// Mitsubishi GX Works2 project: PLC_Group_44   PLC: FX3G

// global labels: Global1
VAR_GLOBAL
  switch7 AT X007 : BOOL;
  lamp7 AT Y007 : BOOL;
  berry_input AT D1100 : INT;
  lemon_input AT D1102 : INT;
  STABILIZER_input AT D1104 : INT;
  GUM_input AT D1106 : INT;
  BERRY_stock AT D1200 : INT;
  LEMON_stock AT D1202 : INT;
  STABILIZER_stock AT D1204 : INT;
  GUM_stock AT D1206 : INT;
  M_start AT M0 : BOOL;
  storage AT D1304 : INT;
  switch5 AT X005 : BOOL;
  analog_input1 AT D8280 : INT;
  switch1 AT X001 : BOOL;
  save_analog_input1 AT D8202 : INT;
END_VAR
VAR_GLOBAL CONSTANT
  K_5 : INT := 2000;
  K_6 : INT := 2400;
  K_10 : INT := 4000;
END_VAR
VAR_GLOBAL
  M_normal AT M1 : BOOL;
  M_pinuk AT M2 : BOOL;
END_VAR
VAR_GLOBAL CONSTANT
  K_7 : INT := 7;
  K_berry_normal : INT := 280;
  K_berry_pinuk : INT := 385;
  K_lemon_normal : INT := 455;
  K_lemon_pinuk : INT := 665;
  K_gum_normal : INT := 28;
  K_gum_pinuk : INT := 70;
  K_stabilizer_normal : INT := 105;
  K_stabilizer_pinuk : INT := 210;
END_VAR
VAR_GLOBAL
  M_exit AT M4 : BOOL;
  BERRY_to_subtract AT D1500 : INT;
  LEMON_to_subtract AT D1502 : INT;
  STABILIZER_to_subtract AT D1504 : INT;
  GUM_to_subtract AT D1506 : INT;
  M_check_stock AT M5 : BOOL;
  M_make_icecream AT M6 : BOOL;
END_VAR
VAR_GLOBAL CONSTANT
  K_berry_total_normal : INT := 350;
  K_berry_total_pinuk : INT := 560;
  K_lemon_total_normal : INT := 490;
  K_lemon_total_pinuk : INT := 700;
END_VAR
VAR_GLOBAL
  BERRY_total AT D1508 : INT;
  LEMON_total AT D1510 : INT;
  making_icecream_timer_c AT TC0 : BOOL;
END_VAR
VAR_GLOBAL CONSTANT
  K_50 : INT := 50;
END_VAR
VAR_GLOBAL
  making_icecream_timer_s AT TS0 : BOOL;
  lamp0 AT Y000 : BOOL;
  M_empty AT M7 : BOOL;
  M_cool_icecream AT M8 : BOOL;
  switch2 AT X002 : BOOL;
  cooling_icecream_timer_c AT TC1 : BOOL;
  cooling_icecream_timer_s AT TS1 : BOOL;
END_VAR
VAR_GLOBAL CONSTANT
  K_80 : INT := 80;
END_VAR
VAR_GLOBAL
  lamp2 AT Y002 : BOOL;
  switch3 AT X003 : BOOL;
  M_mix_materials AT M9 : BOOL;
  M_make_icecream_timer AT M11 : BOOL;
  M_cool_icecream_timer AT M10 : BOOL;
END_VAR
VAR_GLOBAL CONSTANT
  K_mixing_total_normal : INT := 868;
  K_mixing_total_pinuk : INT := 1330;
  K_3 : INT := 3;
END_VAR
VAR_GLOBAL
  mixing_total AT D1512 : INT;
  mixing_duration AT D1514 : INT;
  M_mix_materials_timer AT M12 : BOOL;
  mix_materials_timer_c AT TC2 : BOOL;
  mix_materials_timer_s AT TS2 : BOOL;
  lamp_5_timer_c AT TC3 : BOOL;
  lamp_5_timer_s AT TS3 : BOOL;
  lamp5 AT Y005 : BOOL;
  lamp_6_timer_c AT TC4 : BOOL;
  lamp_6_timer_s AT TS4 : BOOL;
  lamp6 AT Y006 : BOOL;
END_VAR
VAR_GLOBAL CONSTANT
  K_30 : INT := 30;
  K_01 : INT := 40;
  K_0 : INT;
END_VAR
VAR_GLOBAL
  M_BERRY_stock_check AT M14 : BOOL;
  M_LEMON_stock_check AT M15 : BOOL;
  M_STABILIZER_stock_check AT M16 : BOOL;
  M_GUM_stock_check AT M17 : BOOL;
  analog_output AT D8282 : INT;
END_VAR
VAR_GLOBAL CONSTANT
  K_10_timer : INT := 10;
END_VAR
VAR_GLOBAL
  M_cool_and_mix AT M18 : BOOL;
  make_LEMON AT D1308 : INT;
  make_BERRY AT D1306 : INT;
  cool_BERRY AT D1300 : INT;
  cool_LEMON AT D1302 : INT;
  mix_container AT D1310 : INT;
  M_blink_lamps AT M13 : BOOL;
  M_enough_stock AT M3 : BOOL;
END_VAR

// task Task_01 (event TRUE, interval 0, priority 31): POU_01

PROGRAM POU_01
(* structured ladder/FBD written out as ST: instructions are called as NAME(EN, inputs, outputs); _pN, _eN, _tN stand for wires *)
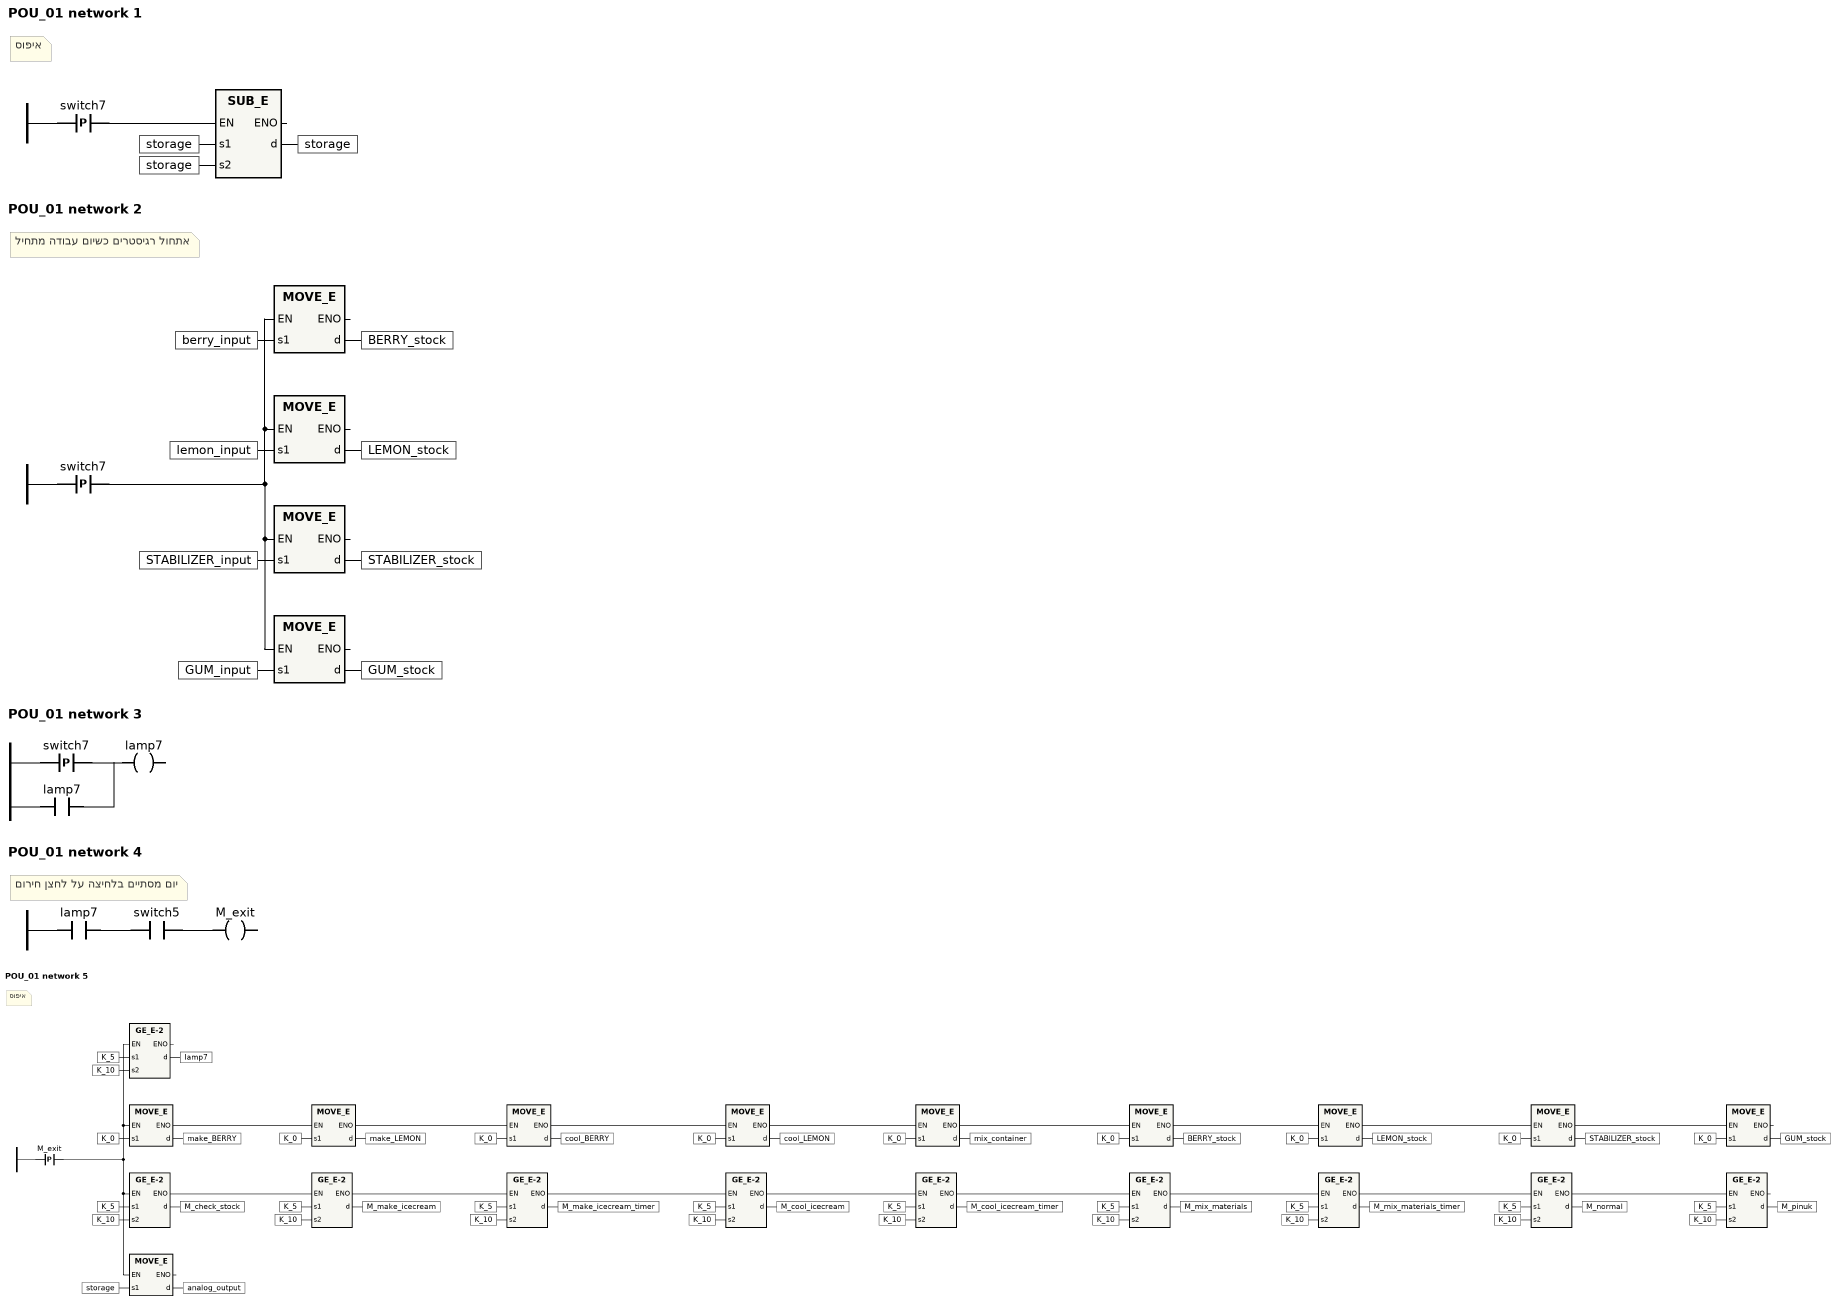
(* network 1 *)
(* איפוס *)
SUB_E(LDP(TRUE, switch7), storage, storage, storage);
(* network 2 *)
(* אתחול רגיסטרים כשיום עבודה מתחיל *)
_p1 := LDP(TRUE, switch7);
MOVE_E(_p1, berry_input, BERRY_stock);
MOVE_E(_p1, lemon_input, LEMON_stock);
MOVE_E(_p1, STABILIZER_input, STABILIZER_stock);
MOVE_E(_p1, GUM_input, GUM_stock);
(* network 3 *)
lamp7 := LDP(TRUE, switch7) OR lamp7;
(* network 4 *)
(* יום מסתיים בלחיצה על לחצן חירום *)
M_exit := lamp7 AND switch5;
(* network 5 *)
(* איפוס *)
_p1 := LDP(TRUE, M_exit);
GE_E(_p1, K_5, K_10, lamp7);
_e2 := MOVE_E(_p1, K_0, make_BERRY);
_e3 := MOVE_E(_e2, K_0, make_LEMON);
_e4 := MOVE_E(_e3, K_0, cool_BERRY);
_e5 := MOVE_E(_e4, K_0, cool_LEMON);
_e6 := MOVE_E(_e5, K_0, mix_container);
_e7 := MOVE_E(_e6, K_0, BERRY_stock);
_e8 := MOVE_E(_e7, K_0, LEMON_stock);
_e9 := MOVE_E(_e8, K_0, STABILIZER_stock);
MOVE_E(_e9, K_0, GUM_stock);
MOVE_E(_p1, storage, analog_output);
_e10 := GE_E(_p1, K_5, K_10, M_check_stock);
_e11 := GE_E(_e10, K_5, K_10, M_make_icecream);
_e12 := GE_E(_e11, K_5, K_10, M_make_icecream_timer);
_e13 := GE_E(_e12, K_5, K_10, M_cool_icecream);
_e14 := GE_E(_e13, K_5, K_10, M_cool_icecream_timer);
_e15 := GE_E(_e14, K_5, K_10, M_mix_materials);
_e16 := GE_E(_e15, K_5, K_10, M_mix_materials_timer);
_e17 := GE_E(_e16, K_5, K_10, M_normal);
GE_E(_e17, K_5, K_10, M_pinuk);
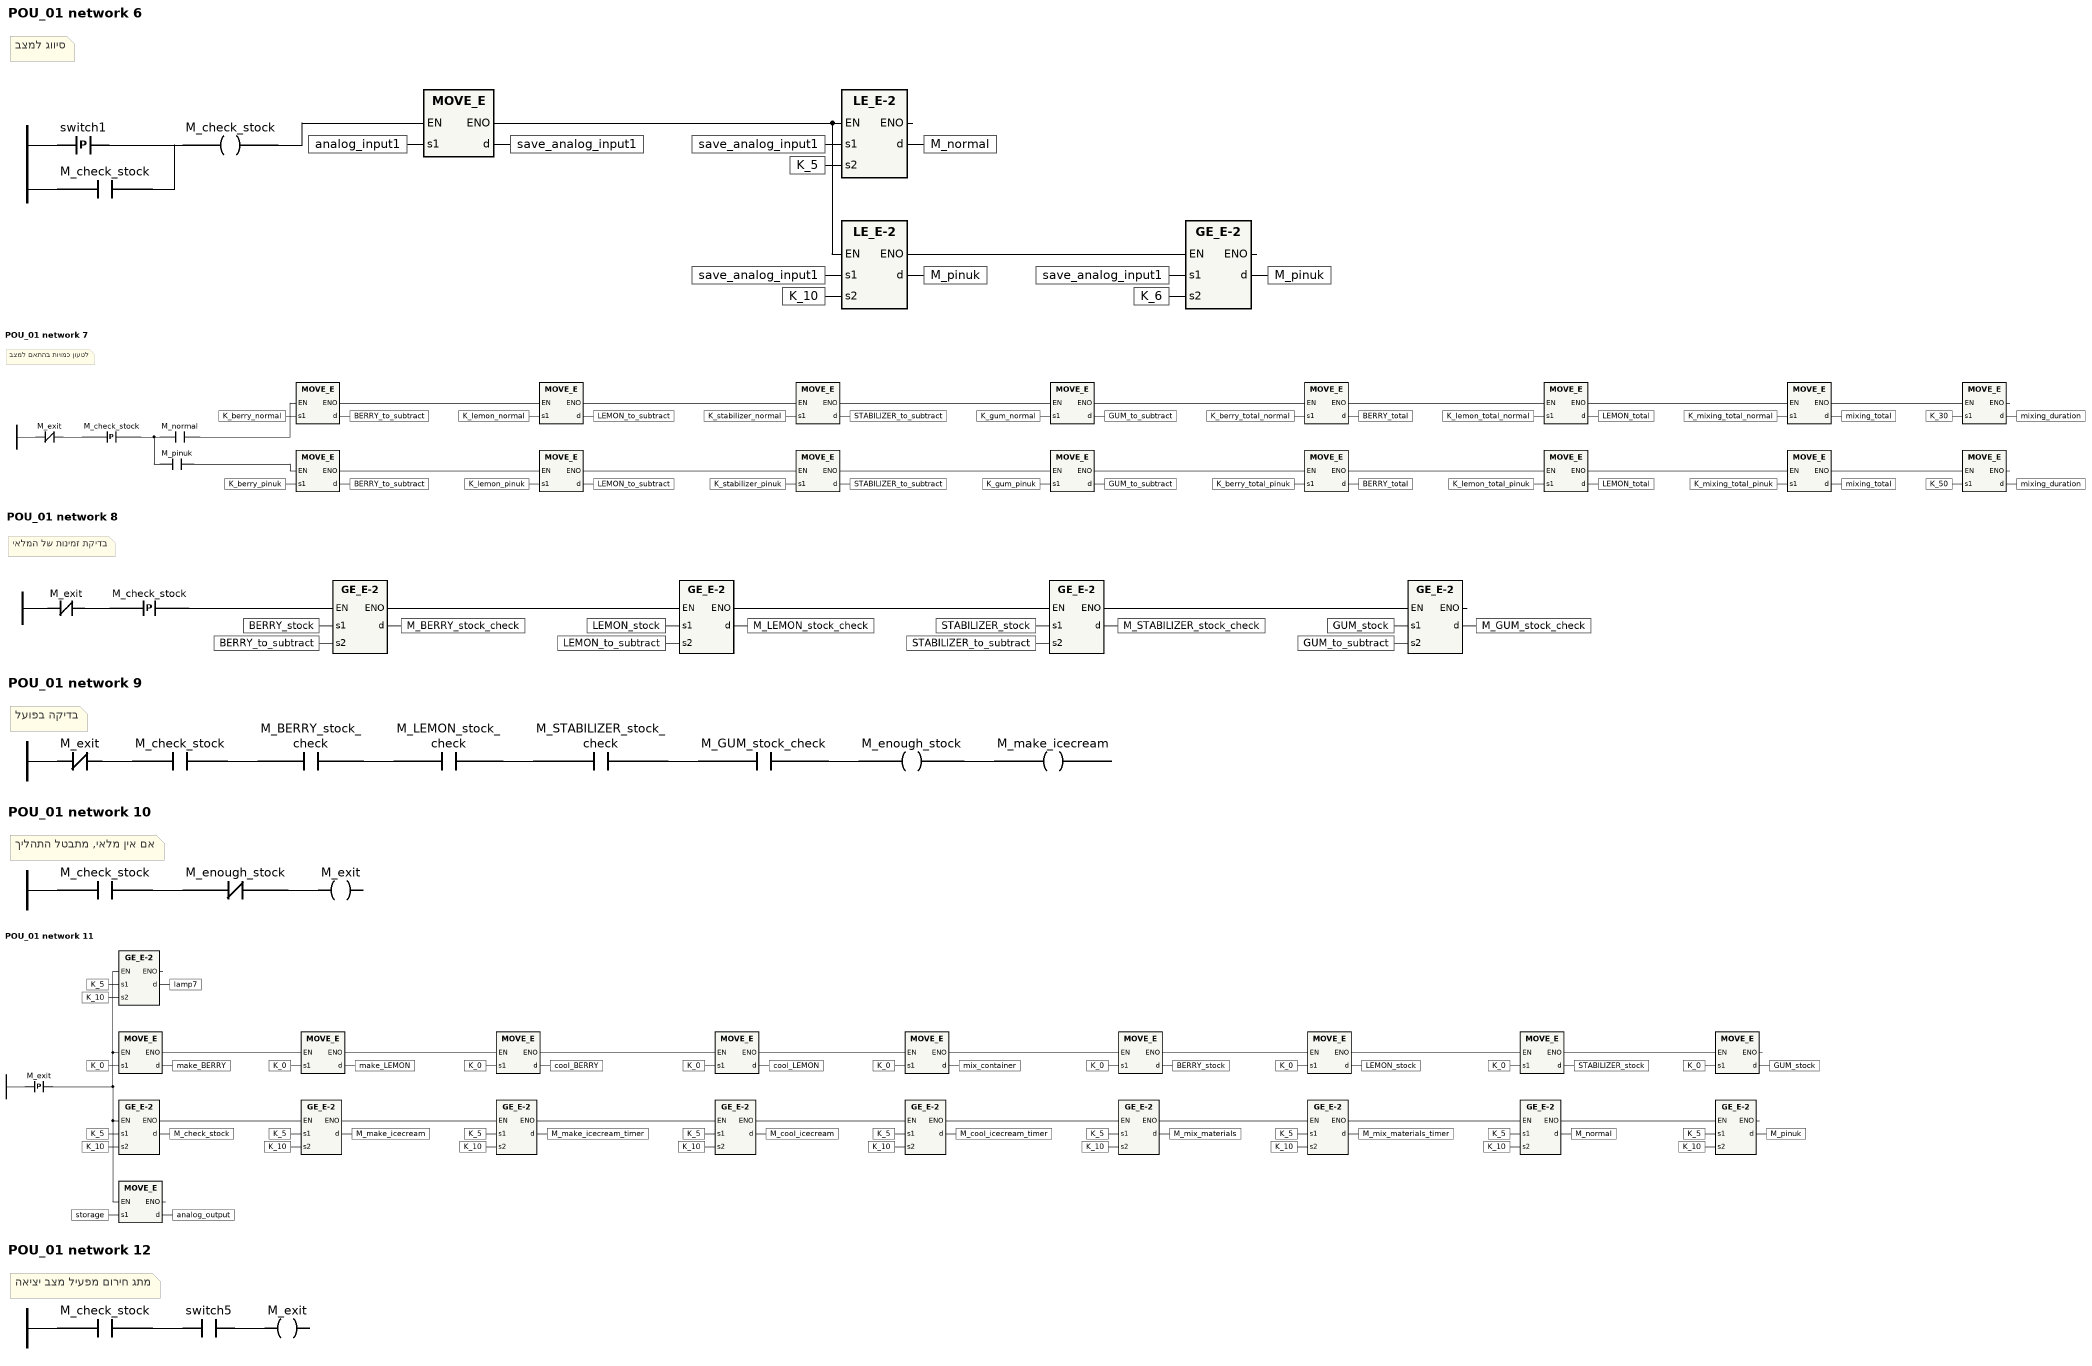
(* network 6 *)
(* סיווג למצב *)
_p1 := LDP(TRUE, switch1) OR M_check_stock;
M_check_stock := _p1;
_e2 := MOVE_E(_p1, analog_input1, save_analog_input1);
LE_E(_e2, save_analog_input1, K_5, M_normal);
_e3 := LE_E(_e2, save_analog_input1, K_10, M_pinuk);
GE_E(_e3, save_analog_input1, K_6, M_pinuk);
(* network 7 *)
(* לטעון כמויות בהתאם למצב *)
_p1 := NOT M_exit AND LDP(TRUE, M_check_stock);
_e2 := MOVE_E(_p1 AND M_normal, K_berry_normal, BERRY_to_subtract);
_e3 := MOVE_E(_e2, K_lemon_normal, LEMON_to_subtract);
_e4 := MOVE_E(_e3, K_stabilizer_normal, STABILIZER_to_subtract);
_e5 := MOVE_E(_e4, K_gum_normal, GUM_to_subtract);
_e6 := MOVE_E(_e5, K_berry_total_normal, BERRY_total);
_e7 := MOVE_E(_e6, K_lemon_total_normal, LEMON_total);
_e8 := MOVE_E(_e7, K_mixing_total_normal, mixing_total);
MOVE_E(_e8, K_30, mixing_duration);
_e9 := MOVE_E(_p1 AND M_pinuk, K_berry_pinuk, BERRY_to_subtract);
_e10 := MOVE_E(_e9, K_lemon_pinuk, LEMON_to_subtract);
_e11 := MOVE_E(_e10, K_stabilizer_pinuk, STABILIZER_to_subtract);
_e12 := MOVE_E(_e11, K_gum_pinuk, GUM_to_subtract);
_e13 := MOVE_E(_e12, K_berry_total_pinuk, BERRY_total);
_e14 := MOVE_E(_e13, K_lemon_total_pinuk, LEMON_total);
_e15 := MOVE_E(_e14, K_mixing_total_pinuk, mixing_total);
MOVE_E(_e15, K_50, mixing_duration);
(* network 8 *)
(* בדיקת זמינות של המלאי *)
_e1 := GE_E(NOT M_exit AND LDP(TRUE, M_check_stock), BERRY_stock, BERRY_to_subtract, M_BERRY_stock_check);
_e2 := GE_E(_e1, LEMON_stock, LEMON_to_subtract, M_LEMON_stock_check);
_e3 := GE_E(_e2, STABILIZER_stock, STABILIZER_to_subtract, M_STABILIZER_stock_check);
GE_E(_e3, GUM_stock, GUM_to_subtract, M_GUM_stock_check);
(* network 9 *)
(* בדיקה בפועל *)
_p1 := NOT M_exit AND M_check_stock AND M_BERRY_stock_check AND M_LEMON_stock_check AND M_STABILIZER_stock_check AND M_GUM_stock_check;
M_enough_stock := _p1;
M_make_icecream := _p1;
(* network 10 *)
(* אם אין מלאי, מתבטל התהליך *)
M_exit := M_check_stock AND NOT M_enough_stock;
(* network 11 *)
_p1 := LDP(TRUE, M_exit);
GE_E(_p1, K_5, K_10, lamp7);
_e2 := MOVE_E(_p1, K_0, make_BERRY);
_e3 := MOVE_E(_e2, K_0, make_LEMON);
_e4 := MOVE_E(_e3, K_0, cool_BERRY);
_e5 := MOVE_E(_e4, K_0, cool_LEMON);
_e6 := MOVE_E(_e5, K_0, mix_container);
_e7 := MOVE_E(_e6, K_0, BERRY_stock);
_e8 := MOVE_E(_e7, K_0, LEMON_stock);
_e9 := MOVE_E(_e8, K_0, STABILIZER_stock);
MOVE_E(_e9, K_0, GUM_stock);
_e10 := GE_E(_p1, K_5, K_10, M_check_stock);
_e11 := GE_E(_e10, K_5, K_10, M_make_icecream);
_e12 := GE_E(_e11, K_5, K_10, M_make_icecream_timer);
_e13 := GE_E(_e12, K_5, K_10, M_cool_icecream);
_e14 := GE_E(_e13, K_5, K_10, M_cool_icecream_timer);
_e15 := GE_E(_e14, K_5, K_10, M_mix_materials);
_e16 := GE_E(_e15, K_5, K_10, M_mix_materials_timer);
_e17 := GE_E(_e16, K_5, K_10, M_normal);
GE_E(_e17, K_5, K_10, M_pinuk);
MOVE_E(_p1, storage, analog_output);
(* network 12 *)
(* מתג חירום מפעיל מצב יציאה *)
M_exit := M_check_stock AND switch5;
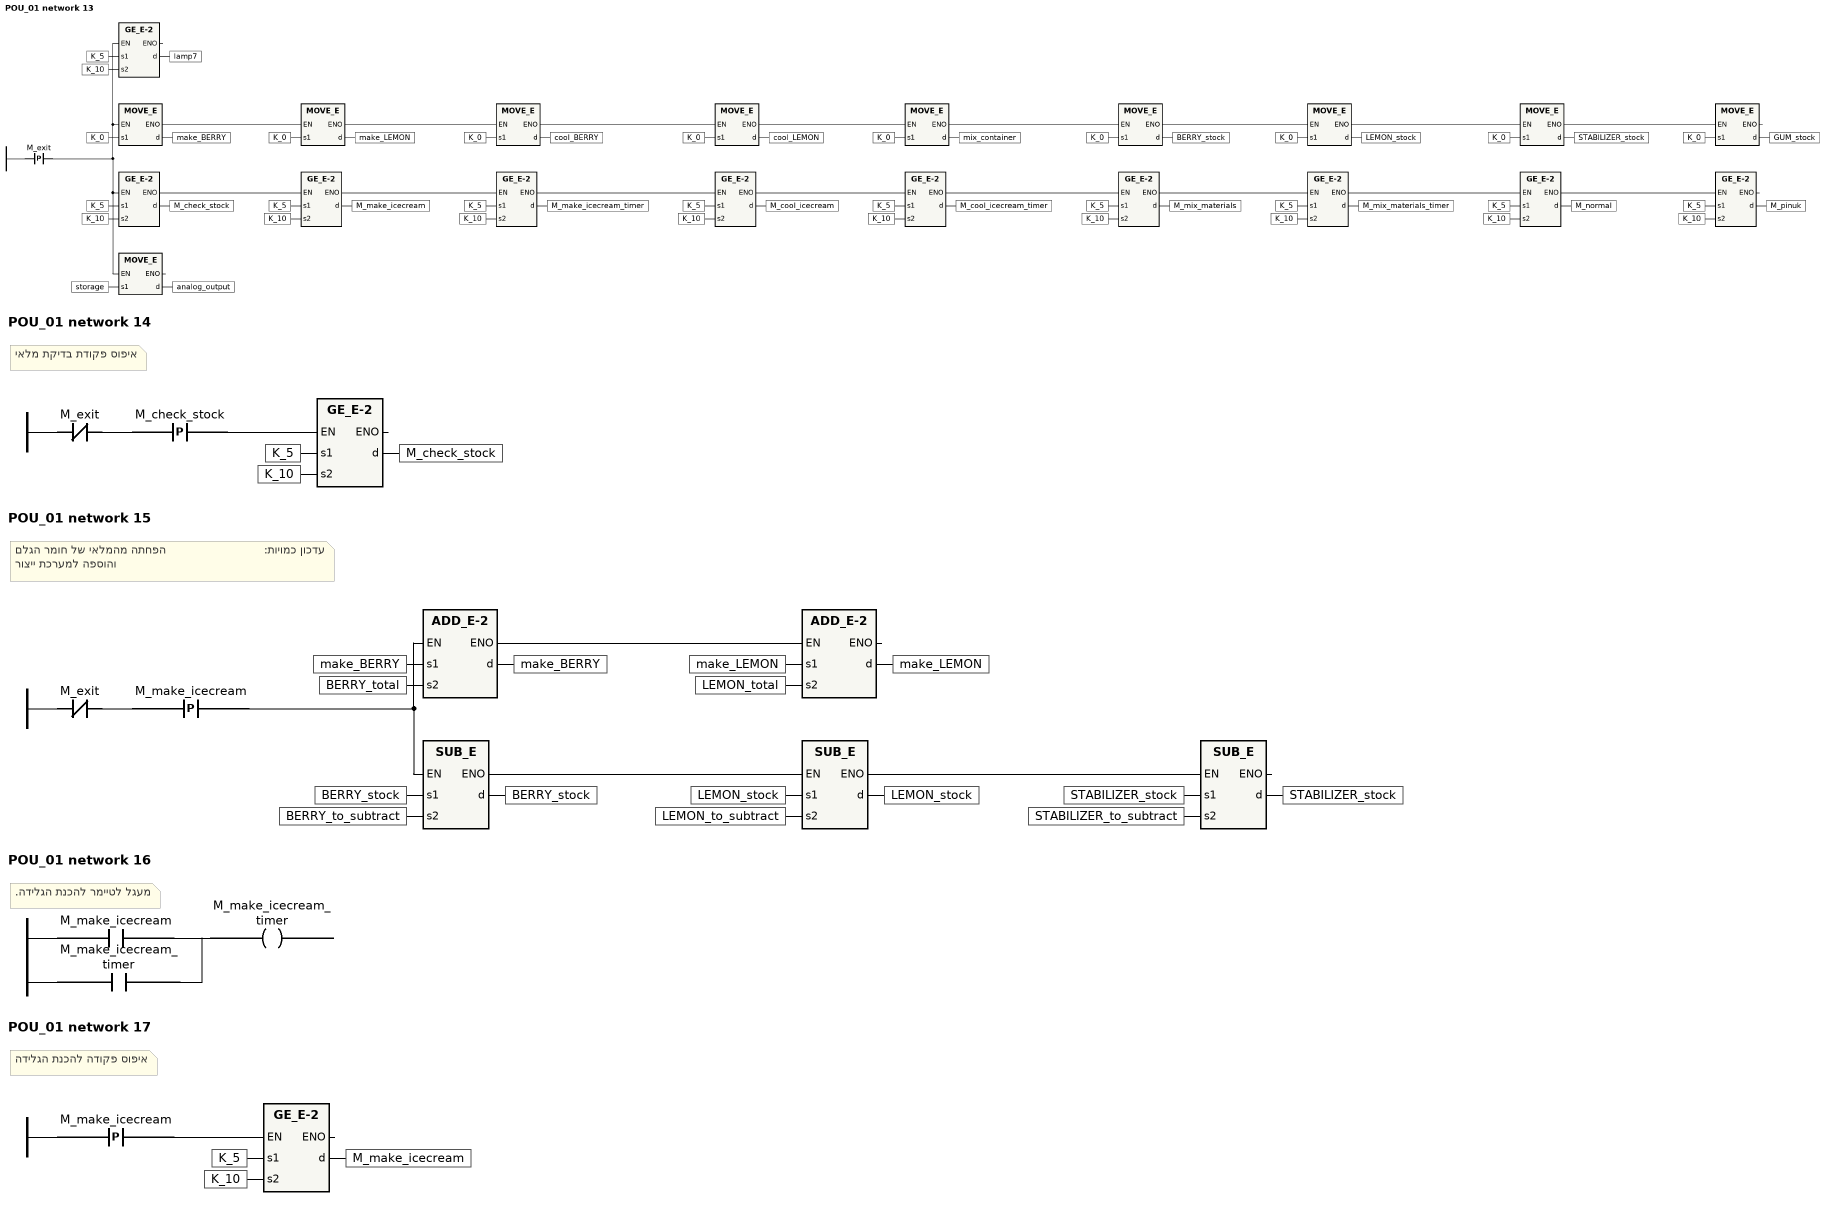
(* network 13 *)
_p1 := LDP(TRUE, M_exit);
GE_E(_p1, K_5, K_10, lamp7);
_e2 := MOVE_E(_p1, K_0, make_BERRY);
_e3 := MOVE_E(_e2, K_0, make_LEMON);
_e4 := MOVE_E(_e3, K_0, cool_BERRY);
_e5 := MOVE_E(_e4, K_0, cool_LEMON);
_e6 := MOVE_E(_e5, K_0, mix_container);
_e7 := MOVE_E(_e6, K_0, BERRY_stock);
_e8 := MOVE_E(_e7, K_0, LEMON_stock);
_e9 := MOVE_E(_e8, K_0, STABILIZER_stock);
MOVE_E(_e9, K_0, GUM_stock);
_e10 := GE_E(_p1, K_5, K_10, M_check_stock);
_e11 := GE_E(_e10, K_5, K_10, M_make_icecream);
_e12 := GE_E(_e11, K_5, K_10, M_make_icecream_timer);
_e13 := GE_E(_e12, K_5, K_10, M_cool_icecream);
_e14 := GE_E(_e13, K_5, K_10, M_cool_icecream_timer);
_e15 := GE_E(_e14, K_5, K_10, M_mix_materials);
_e16 := GE_E(_e15, K_5, K_10, M_mix_materials_timer);
_e17 := GE_E(_e16, K_5, K_10, M_normal);
GE_E(_e17, K_5, K_10, M_pinuk);
MOVE_E(_p1, storage, analog_output);
(* network 14 *)
(* איפוס פקודת בדיקת מלאי *)
GE_E(NOT M_exit AND LDP(TRUE, M_check_stock), K_5, K_10, M_check_stock);
(* network 15 *)
(* עדכון כמויות:                            הפחתה מהמלאי של חומר הגלם והוספה למערכת ייצור *)
_p1 := NOT M_exit AND LDP(TRUE, M_make_icecream);
_e2 := ADD_E(_p1, make_BERRY, BERRY_total, make_BERRY);
ADD_E(_e2, make_LEMON, LEMON_total, make_LEMON);
_e3 := SUB_E(_p1, BERRY_stock, BERRY_to_subtract, BERRY_stock);
_e4 := SUB_E(_e3, LEMON_stock, LEMON_to_subtract, LEMON_stock);
SUB_E(_e4, STABILIZER_stock, STABILIZER_to_subtract, STABILIZER_stock);
(* network 16 *)
(* מעגל לטיימר להכנת הגלידה. *)
M_make_icecream_timer := M_make_icecream OR M_make_icecream_timer;
(* network 17 *)
(* איפוס פקודה להכנת הגלידה *)
GE_E(LDP(TRUE, M_make_icecream), K_5, K_10, M_make_icecream);
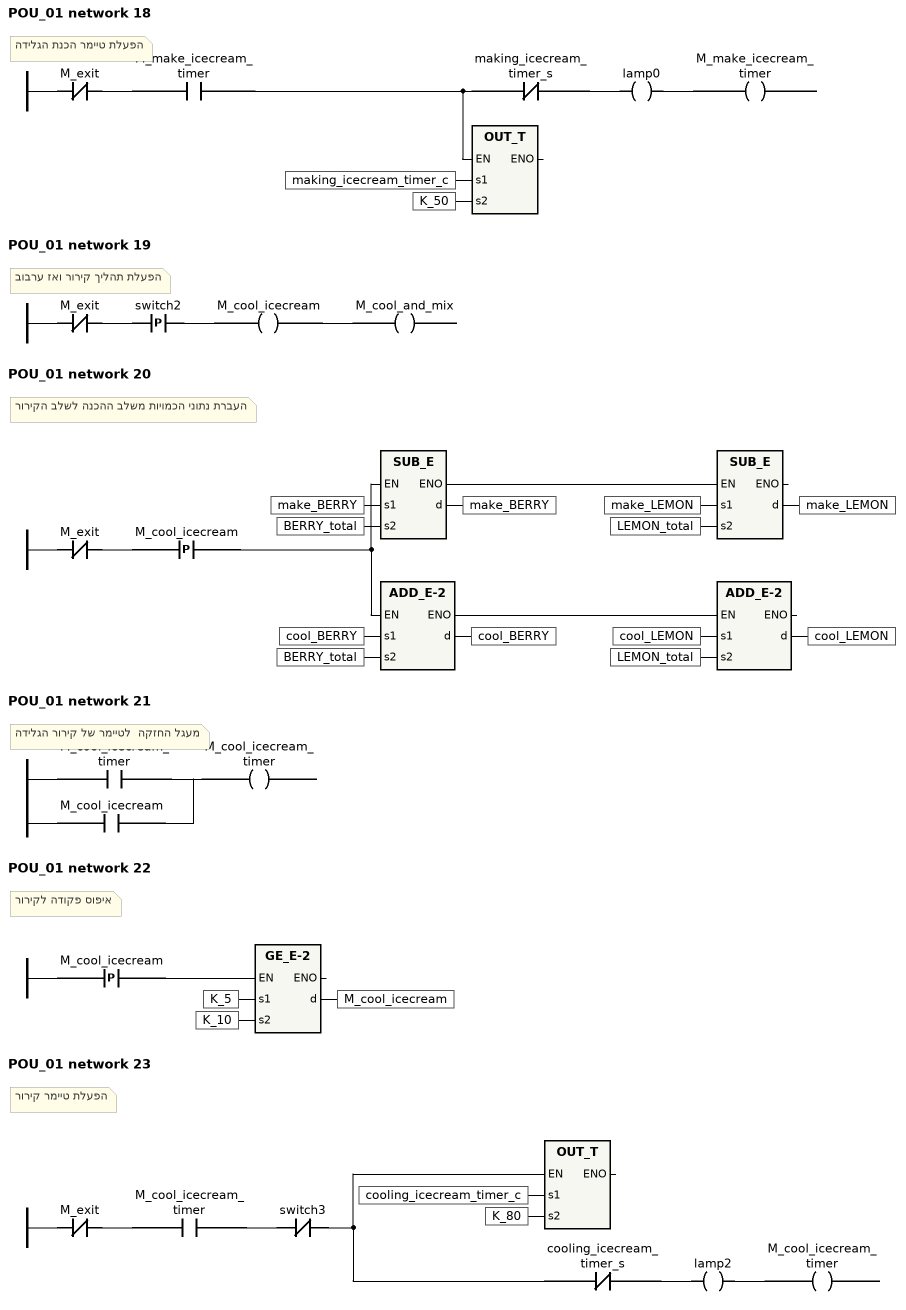
(* network 18 *)
(* הפעלת טיימר הכנת הגלידה *)
_p1 := NOT M_exit AND M_make_icecream_timer;
_p2 := _p1 AND NOT making_icecream_timer_s;
lamp0 := _p2;
M_make_icecream_timer := _p2;
OUT_T(_p1, making_icecream_timer_c, K_50);
(* network 19 *)
(* הפעלת תהליך קירור ואז ערבוב *)
_p1 := NOT M_exit AND LDP(TRUE, switch2);
M_cool_icecream := _p1;
M_cool_and_mix := _p1;
(* network 20 *)
(* העברת נתוני הכמויות משלב ההכנה לשלב הקירור *)
_p1 := NOT M_exit AND LDP(TRUE, M_cool_icecream);
_e2 := SUB_E(_p1, make_BERRY, BERRY_total, make_BERRY);
SUB_E(_e2, make_LEMON, LEMON_total, make_LEMON);
_e3 := ADD_E(_p1, cool_BERRY, BERRY_total, cool_BERRY);
ADD_E(_e3, cool_LEMON, LEMON_total, cool_LEMON);
(* network 21 *)
(* מעגל החזקה  לטיימר של קירור הגלידה *)
M_cool_icecream_timer := M_cool_icecream_timer OR M_cool_icecream;
(* network 22 *)
(* איפוס פקודה לקירור *)
GE_E(LDP(TRUE, M_cool_icecream), K_5, K_10, M_cool_icecream);
(* network 23 *)
(* הפעלת טיימר קירור *)
_p1 := NOT M_exit AND M_cool_icecream_timer AND NOT switch3;
OUT_T(_p1, cooling_icecream_timer_c, K_80);
_p2 := _p1 AND NOT cooling_icecream_timer_s;
lamp2 := _p2;
M_cool_icecream_timer := _p2;
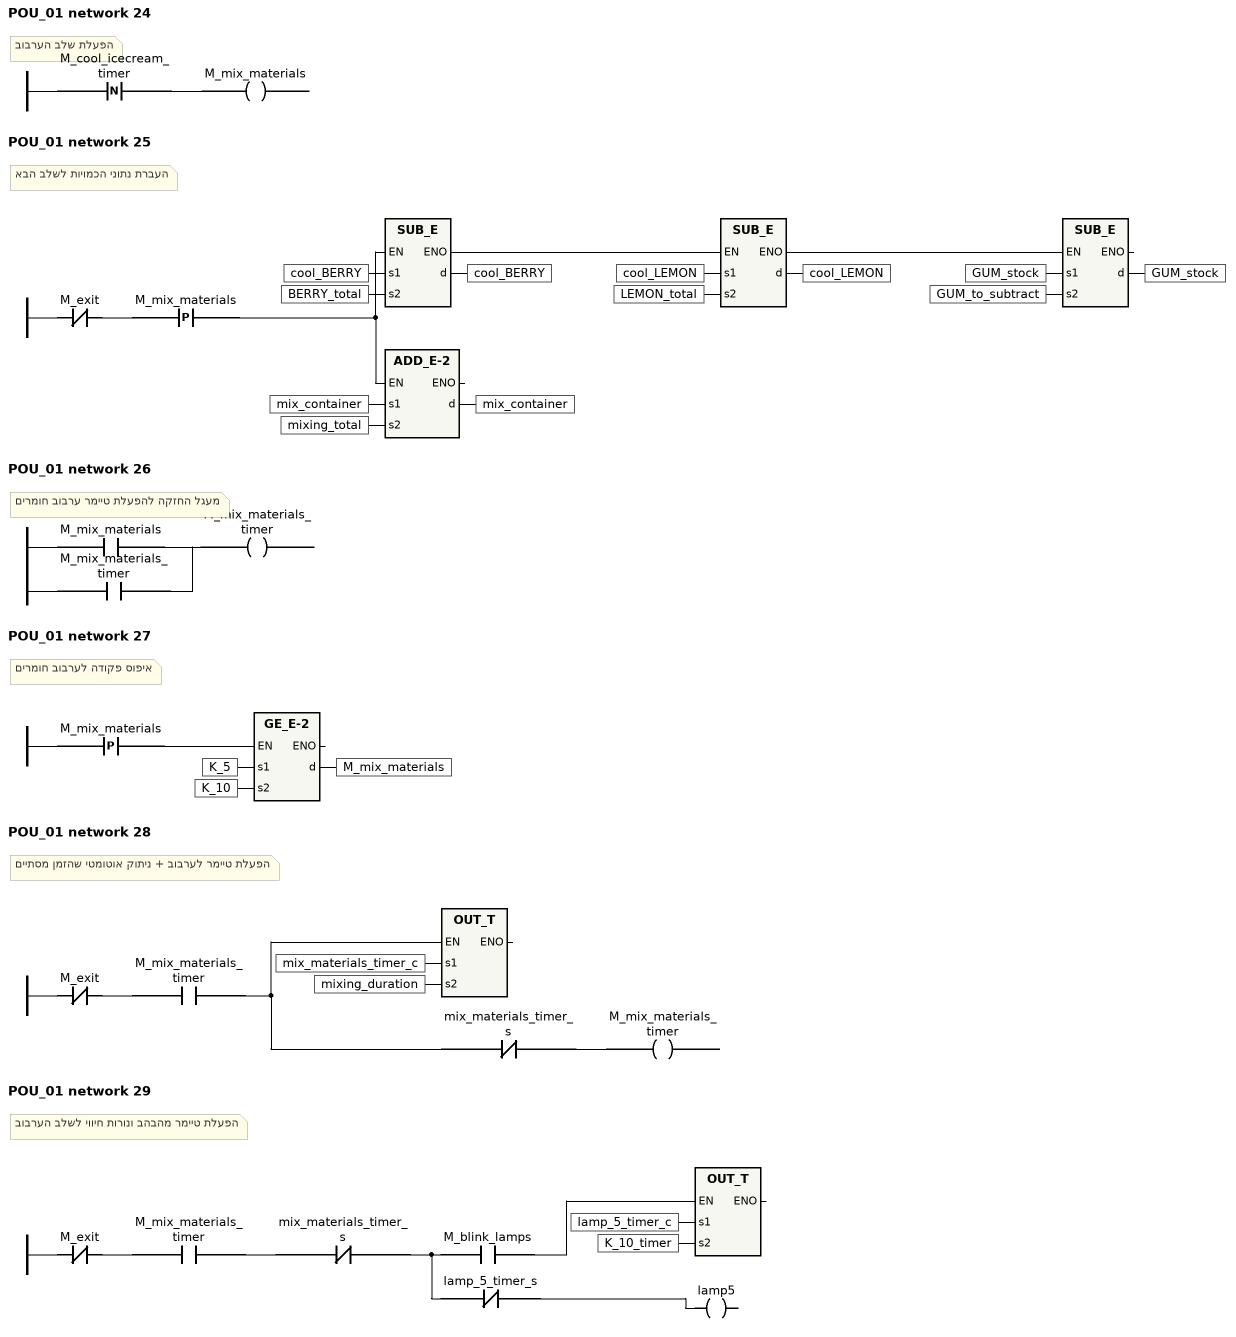
(* network 24 *)
(* הפעלת שלב הערבוב *)
M_mix_materials := LDF(TRUE, M_cool_icecream_timer);
(* network 25 *)
(* העברת נתוני הכמויות לשלב הבא *)
_p1 := NOT M_exit AND LDP(TRUE, M_mix_materials);
_e2 := SUB_E(_p1, cool_BERRY, BERRY_total, cool_BERRY);
_e3 := SUB_E(_e2, cool_LEMON, LEMON_total, cool_LEMON);
SUB_E(_e3, GUM_stock, GUM_to_subtract, GUM_stock);
ADD_E(_p1, mix_container, mixing_total, mix_container);
(* network 26 *)
(* מעגל החזקה להפעלת טיימר ערבוב חומרים *)
M_mix_materials_timer := M_mix_materials OR M_mix_materials_timer;
(* network 27 *)
(* איפוס פקודה לערבוב חומרים *)
GE_E(LDP(TRUE, M_mix_materials), K_5, K_10, M_mix_materials);
(* network 28 *)
(* הפעלת טיימר לערבוב + ניתוק אוטומטי שהזמן מסתיים *)
_p1 := NOT M_exit AND M_mix_materials_timer;
OUT_T(_p1, mix_materials_timer_c, mixing_duration);
M_mix_materials_timer := _p1 AND NOT mix_materials_timer_s;
(* network 29 *)
(* הפעלת טיימר מהבהב ונורות חיווי לשלב הערבוב *)
_p1 := NOT M_exit AND M_mix_materials_timer AND NOT mix_materials_timer_s;
OUT_T(_p1 AND M_blink_lamps, lamp_5_timer_c, K_10_timer);
lamp5 := _p1 AND NOT lamp_5_timer_s;
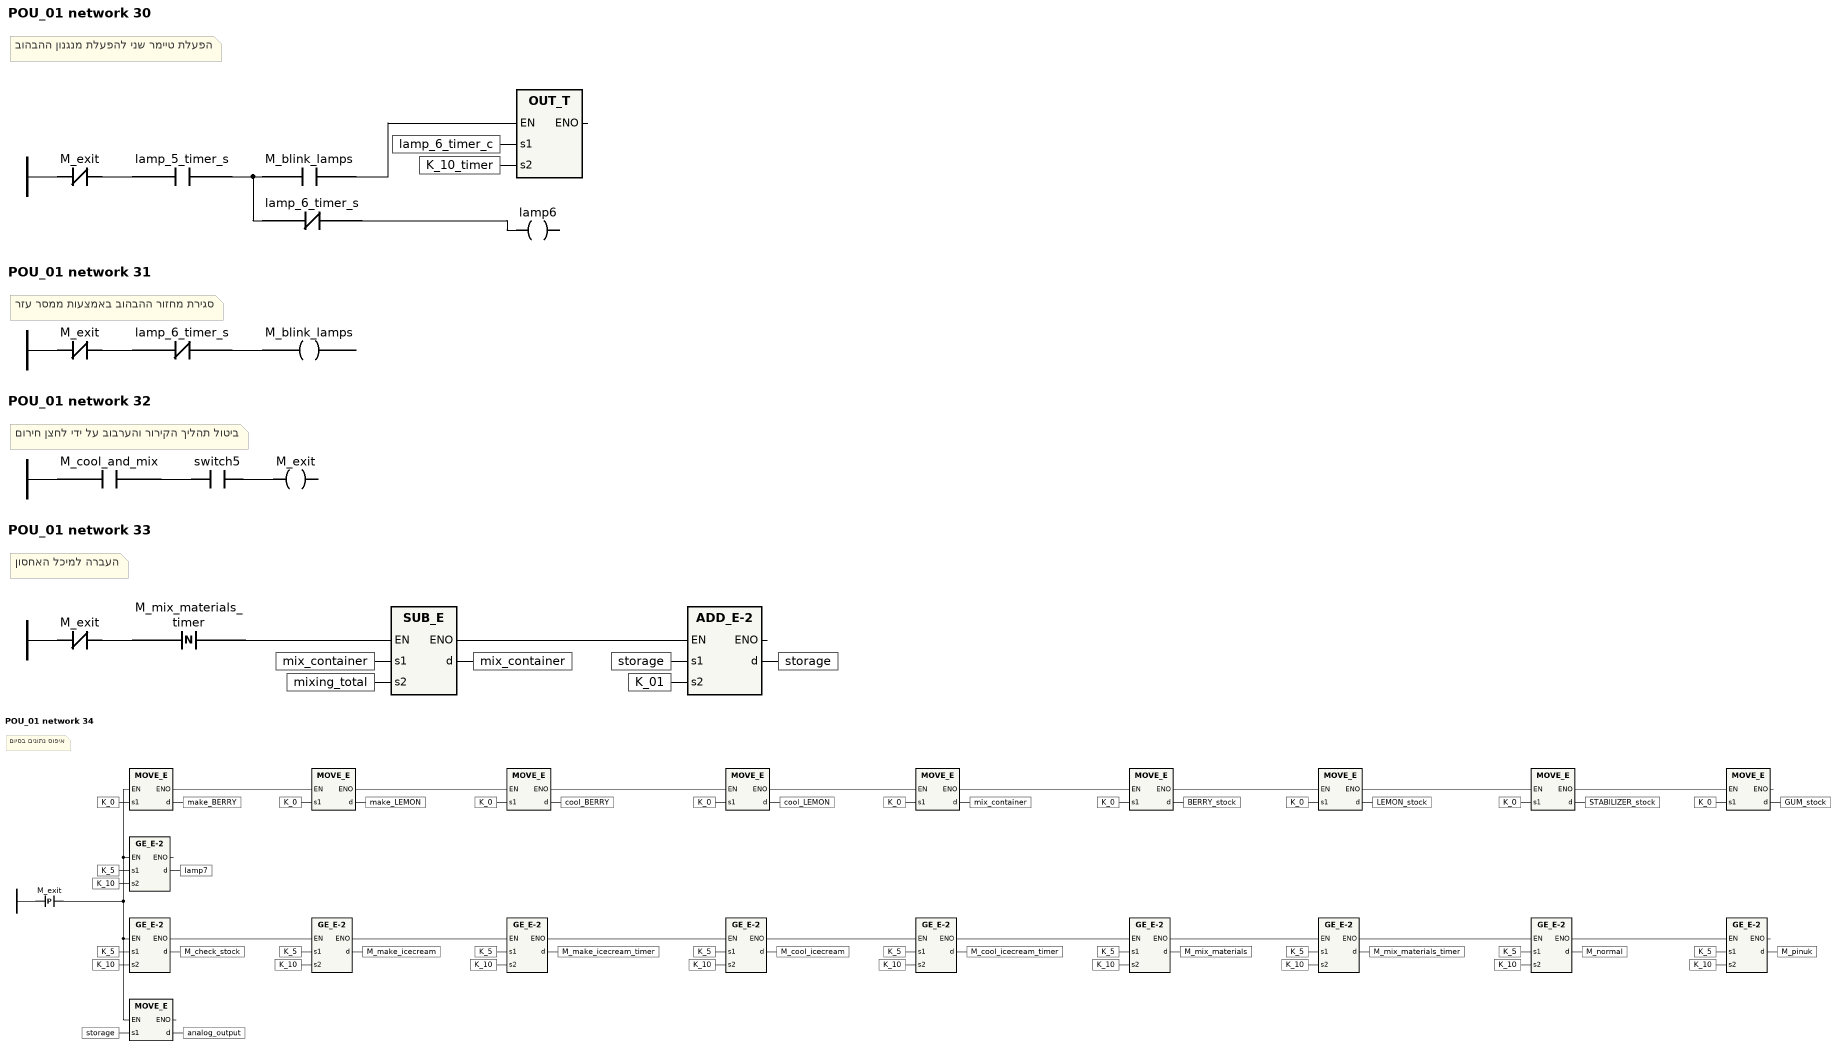
(* network 30 *)
(* הפעלת טיימר שני להפעלת מנגנון ההבהוב *)
_p1 := NOT M_exit AND lamp_5_timer_s;
OUT_T(_p1 AND M_blink_lamps, lamp_6_timer_c, K_10_timer);
lamp6 := _p1 AND NOT lamp_6_timer_s;
(* network 31 *)
(* סגירת מחזור ההבהוב באמצעות ממסר עזר *)
M_blink_lamps := NOT M_exit AND NOT lamp_6_timer_s;
(* network 32 *)
(* ביטול תהליך הקירור והערבוב על ידי לחצן חירום *)
M_exit := M_cool_and_mix AND switch5;
(* network 33 *)
(* העברה למיכל האחסון *)
_e1 := SUB_E(NOT M_exit AND LDF(TRUE, M_mix_materials_timer), mix_container, mixing_total, mix_container);
ADD_E(_e1, storage, K_01, storage);
(* network 34 *)
(* איפוס נתונים בסיום *)
_p1 := LDP(TRUE, M_exit);
_e2 := MOVE_E(_p1, K_0, make_BERRY);
_e3 := MOVE_E(_e2, K_0, make_LEMON);
_e4 := MOVE_E(_e3, K_0, cool_BERRY);
_e5 := MOVE_E(_e4, K_0, cool_LEMON);
_e6 := MOVE_E(_e5, K_0, mix_container);
_e7 := MOVE_E(_e6, K_0, BERRY_stock);
_e8 := MOVE_E(_e7, K_0, LEMON_stock);
_e9 := MOVE_E(_e8, K_0, STABILIZER_stock);
MOVE_E(_e9, K_0, GUM_stock);
GE_E(_p1, K_5, K_10, lamp7);
_e10 := GE_E(_p1, K_5, K_10, M_check_stock);
_e11 := GE_E(_e10, K_5, K_10, M_make_icecream);
_e12 := GE_E(_e11, K_5, K_10, M_make_icecream_timer);
_e13 := GE_E(_e12, K_5, K_10, M_cool_icecream);
_e14 := GE_E(_e13, K_5, K_10, M_cool_icecream_timer);
_e15 := GE_E(_e14, K_5, K_10, M_mix_materials);
_e16 := GE_E(_e15, K_5, K_10, M_mix_materials_timer);
_e17 := GE_E(_e16, K_5, K_10, M_normal);
GE_E(_e17, K_5, K_10, M_pinuk);
MOVE_E(_p1, storage, analog_output);
END_PROGRAM
